(* PLC project Prueba, adfadsf asdfasdfadsf 1 *)
(* stored: creationDateTime 2011-11-03T09:53:23, modificationDateTime 2011-11-03T10:05:25 *)

FUNCTION_BLOCK sfc1
  VAR
    FCB : BOOL;
  END_VAR

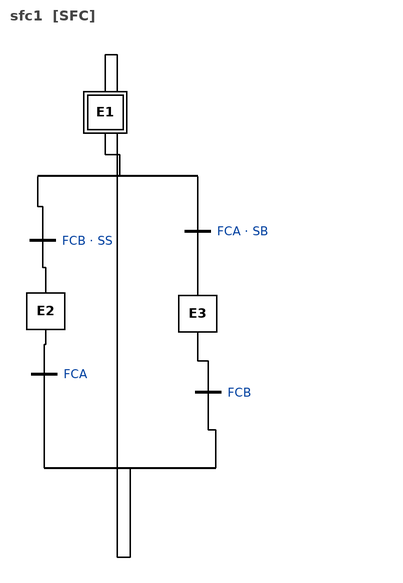
INITIAL_STEP E1:
END_STEP
TRANSITION FROM E1 TO E2
  := FCB · SS;
END_TRANSITION
TRANSITION FROM E1 TO E3
  := FCA · SB;
END_TRANSITION
STEP E2:
END_STEP
TRANSITION FROM E2 TO E1
  := FCA;
END_TRANSITION
STEP E3:
END_STEP
TRANSITION FROM E3 TO E1
  := FCB;
END_TRANSITION
END_FUNCTION_BLOCK
